DATA_BLOCK "KistlerPresser2_DB"
{ S7_Optimized_Access := 'FALSE' }
VERSION : 0.1
NON_RETAIN
// ATTRIBUTES
// AUTO_NUMBER = False
// BLOCK_NUMBER = 2322
// END_ATTRIBUTES
   STRUCT
      ShaftID : Array[0..50] of Char;
      HousingID_1 : Array[0..50] of Char;
      HousingID_2 : Array[0..50] of Char;
      Shaft : String[48];
      spare : String[48];
   END_STRUCT;


BEGIN
   spare := '46';

END_DATA_BLOCK

